// TIA Portal V15 export
// export: Created 2019-01-09T10:35:33.7952885Z, ExportSetting WithDefaults, WithReadOnly, DisplayName Totally Integrated Automation Portal, DisplayVersion V15 Update 2, DisplayName TIA Portal Openness, DisplayVersion V15 Update 2, DisplayName STEP 7 Professional, DisplayVersion V15 Update 2, DisplayName STEP 7 Safety, DisplayVersion V15, DisplayName WinCC Professional, DisplayVersion V15 Update 2, DisplayName SIMATIC Visualization Architect, DisplayVersion V15 Update 1
DATA_BLOCK "FGDB_DESK_NAME"   // DB49
TITLE = Control desk area 10 / Steuerung Pultbereich 10
{ S7_Optimized_Access := 'FALSE' }
AUTHOR : integra
FAMILY : BS
VERSION : 0.5
// stored: AutoNumber true, CodeModifiedDate 2018-01-29T16:41:28.5619003Z, CompileDate 2018-02-20T10:24:34.845539Z, CreationDate 2016-12-16T08:19:30.2842824Z, DBAccessibleFromOPCUA true, InstanceOfName iFG_DESK, InstanceOfNumber 1018, InstanceOfType FB, InterfaceModifiedDate 2018-01-29T16:41:25.4524836Z, IsConsistent true, IsKnowHowProtected false, ModifiedDate 2018-01-29T16:41:28.5619003Z, ParameterModified 2018-01-24T11:29:10.7847282Z, StructureModified 2018-01-24T11:29:10.7847282Z, UDAEnableTagReadback false
"iFG_DESK"
   // VAR_INPUT
   //    desk : Int;
   //    fct : Int;
   //    setup : Bool;
   //    auto : Bool;
   //    autoStart : Bool;
   //    autoEnd : Bool;
   //    enableIn : Bool;
   //    ack : Bool;
   //    lampTest : Bool;
   //    startupWarning : Bool;
   //    autoStartFromSection : Bool;
   // END_VAR
   // VAR_OUTPUT
   //    setupOn : Bool;
   //    automaticOn : Bool;
   //    setupLamp : Bool;
   //    automaticLamp : Bool;
   //    eStopLamp : Bool;
   //    faultLamp : Bool;
   //    automaticStartup : Bool;
   //    fault : Bool;
   //    faultExt : Bool;
   // END_VAR
   // VAR RETAIN
   //    idx : Int;
   //    sectionnumber : Int;
   //    desknumber : Int;
   //    stationnumber : Int;
   //    dbnumber : Int;
   //    function : Int;
   //    numberInternalMessages : Int;
   //    numberExternalMessages : Int;
   //    F : Struct
   //       fct : Bool;
   //    END_STRUCT;
   //    "M" : Struct
   //       noAuto : Bool;
   //       noAutoExtern : Bool;
   //    END_STRUCT;
   //    Masks : Struct
   //       disableFault_1_8 : Byte;
   //       prodRelevantFault1_8 : Byte;
   //    END_STRUCT;
   //    LastState : Struct
   //       fault_1_8 : Byte;
   //       message_1_8 : Byte;
   //    END_STRUCT;
   //    IfcFGExternal : "iUDT_IFC_SYS_EXTERNAL_ALARM";
   //    Tmr : Struct
   //       s_1 { S7_SetPoint := 'True'} : Int;
   //       a_1 : Int;
   //       s_2 { S7_SetPoint := 'True'} : Int;
   //       a_2 : Int;
   //       s_3 { S7_SetPoint := 'True'} : Int;
   //       a_3 : Int;
   //    END_STRUCT;
   //    StM : Struct
   //       fault : Bool;
   //       setup : Bool;
   //       auto : Bool;
   //       warning : Bool;
   //       eStop : Bool;
   //       safetyStop : Bool;
   //       enableIn : Bool;
   //       enableOutForward : Bool;
   //       enableOutBackward : Bool;
   //       faultPr : Bool;
   //       pairMon : Bool;
   //       specialMode : Bool;
   //       "13" : Bool;
   //       "14" : Bool;
   //       "15" : Bool;
   //       "16" : Bool;
   //       "17" : Bool;
   //       "18" : Bool;
   //       "19" : Bool;
   //       "20" : Bool;
   //       "21" : Bool;
   //       "22" : Bool;
   //       "23" : Bool;
   //       "24" : Bool;
   //       "25" : Bool;
   //       "26" : Bool;
   //       "27" : Bool;
   //       "28" : Bool;
   //       "29" : Bool;
   //       "30" : Bool;
   //       "31" : Bool;
   //       "32" : Bool;
   //    END_STRUCT;
   //    VB : Struct
   //       fault : Bool;
   //       setup : Bool;
   //       auto : Bool;
   //       warning : Bool;
   //       eStop : Bool;
   //       safetyStop : Bool;
   //       enableIn : Bool;
   //       enableOutForward : Bool;
   //       enableOutBackward : Bool;
   //       faultPr : Bool;
   //       pairMon : Bool;
   //       specialMode : Bool;
   //       "13" : Bool;
   //       "14" : Bool;
   //       "15" : Bool;
   //       "16" : Bool;
   //       "17" : Bool;
   //       "18" : Bool;
   //       "19" : Bool;
   //       "20" : Bool;
   //       "21" : Bool;
   //       "22" : Bool;
   //       "23" : Bool;
   //       "24" : Bool;
   //       "25" : Bool;
   //       "26" : Bool;
   //       "27" : Bool;
   //       "28" : Bool;
   //       "29" : Bool;
   //       "30" : Bool;
   //       "31" : Bool;
   //       "32" : Bool;
   //    END_STRUCT;
   //    VCB : Struct
   //       ack : Bool;
   //       ackDesk : Bool;
   //    END_STRUCT;
   //    TmrB : Struct
   //       "1_Enable" : Bool;
   //       "1_Run" : Bool;
   //       "1_Done" : Bool;
   //       "2_Enable" : Bool;
   //       "2_Run" : Bool;
   //       "2_Done" : Bool;
   //       "3_Enable" : Bool;
   //       "3_Run" : Bool;
   //       "3_Done" : Bool;
   //    END_STRUCT;
   //    D : Struct
   //       enableIn : Bool;
   //       visuAck : Bool;
   //       visuAckDesk : Bool;
   //       auxEnableIn : Bool;
   //       operatingModeMemory : Bool;
   //       operatingModeMemoryRd : Bool;
   //       deskSetup : Bool;
   //       deskAutomaticPosition : Bool;
   //       deskAutomatic : Bool;
   //       auxDeskAutomaticPosition : Bool;
   //       fPLampTest : Bool;
   //       pPLampTest : Bool;
   //       fPAutoStart : Bool;
   //       pPAutoStart : Bool;
   //       fpAck : Bool;
   //       pPAck : Bool;
   //       autoStartFromSection : Bool;
   //       fpControlVoltageOn : Bool;
   //    END_STRUCT;
   //    V : Struct
   //       runtime : UInt;
   //    END_STRUCT;
   //    ifcDesk { ExternalAccessible := 'False'; ExternalVisible := 'False'; ExternalWritable := 'False'} : "iUDT_IFC_DESK";
   // END_VAR
BEGIN
END_DATA_BLOCK
